// TIA Portal V18 export
TYPE "UDT_RECIPE"
   STRUCT
      TypeName : String[50] := 'Product_1';   // System Defined=
      TypeID : USInt := 1;   // System define= product type for parameters of servo ,press and so on
      FixtureID : Array[1..16] of Byte;
      A1_TableFixtureCode : Array[0..10] of String[128];   // 激光刻印程序号
      A2_TableFixtureCode : Array[0..10] of String[128];   // 贴标10号垂直气缸是否去工作位
      A1RingUnloadingFixtureCode : String[128] := 'SZ23055-OP010-E-Compresspr-ring1 cutting tool';
      E1LoadingNGFixtureCode : String[128] := 'SZ23055-OP010-E-Compressor-Left NG tooling-1';
      ShaftScanFixtureCode : String[128] := 'SZ23055-OP010-E-Compressor-shaft Rotating scanning tooling-1';
      B1PressFixtureCode : String[128] := 'SZ23055-OP010-E-Compressor-ring1 Below Positioning fixture -1';
      CGlueFixtureCode : String[128] := 'SZ23055-OP010-E-Compressor-Point adhesive tooling-1';
      B1PressCylFixtureCode : String[128] := 'SZ23055-OP010-E-Compressor-ring1 Upper pressing fixture-1';
      A2RingUnloadingFixtureCode : String[128] := 'SZ23055-OP010-E-Compresspr-ring2 cutting tool';
      E2UnloadingNGFixtureCode : String[128] := 'SZ23055-OP010-E-Compressor-Right NG tooling-1';
      B2PressFixtureCode : String[128] := 'SZ23055-OP010-E-Compressor-ring2 Below Positioning fixture -1';
      CGlueNGFixtureCode : String[128] := 'SZ23055-OP010-E-Compressor-NG middle shift tooling-1';
      B2PressCylFixtureCode : String[128] := 'SZ23055-OP010-E-Compressor-ring2 Upper pressing fixture-1';
      R1GripperFixtureCode : Array[1..4] of String[128];
      R2GripperFixtureCode : Array[1..4] of String[128];
      R3GripperFixtureCode : Array[1..4] of String[128];
      B1PressProgram : Int := 1;
      B2PressProgram : Int := 1;
      CGlueShaftIV3Program_1 : Word := 16#0001;
      CGlueShaftIV3Program_2 : Word := 16#0002;
      CGlueShaftIV3Program_3 : Word := 16#0003;
      CGlueShaftIV3Program_4 : Word := 16#0004;
      CGlueMagnetIV3Program : Word := 16#0001;
      CGlueProgram : Int := 1;
   END_STRUCT;
   // FixtureID[1] := 16#00;   // 工装编号
   // FixtureID[2..16] := 16#00;
   // A1_TableFixtureCode[0] := '';
   // A1_TableFixtureCode[1] := 'SZ23055-OP010-E-Compressor-ring1 Loading tooling-1';
   // A1_TableFixtureCode[2] := 'SZ23055-OP010-E-Compressor-ring1 Loading tooling-2';
   // A1_TableFixtureCode[3] := 'SZ23055-OP010-E-Compressor-ring1 Loading tooling-3';
   // A1_TableFixtureCode[4] := 'SZ23055-OP010-E-Compressor-ring1 Loading tooling-4';
   // A1_TableFixtureCode[5] := 'SZ23055-OP010-E-Compressor-ring1 Loading tooling-5';
   // A1_TableFixtureCode[6] := 'SZ23055-OP010-E-Compressor-ring1 Loading tooling-6';
   // A1_TableFixtureCode[7] := 'SZ23055-OP010-E-Compressor-ring1 Loading tooling-7';
   // A1_TableFixtureCode[8] := 'SZ23055-OP010-E-Compressor-ring1 Loading tooling-8';
   // A1_TableFixtureCode[9..10] := '';
   // A2_TableFixtureCode[0] := '';
   // A2_TableFixtureCode[1] := 'SZ23055-OP010-E-Compressor-ring2 Loading tooling-1';
   // A2_TableFixtureCode[2] := 'SZ23055-OP010-E-Compressor-ring2 Loading tooling-2';
   // A2_TableFixtureCode[3] := 'SZ23055-OP010-E-Compressor-ring2 Loading tooling-3';
   // A2_TableFixtureCode[4] := 'SZ23055-OP010-E-Compressor-ring2 Loading tooling-4';
   // A2_TableFixtureCode[5] := 'SZ23055-OP010-E-Compressor-ring2 Loading tooling-5';
   // A2_TableFixtureCode[6] := 'SZ23055-OP010-E-Compressor-ring2 Loading tooling-6';
   // A2_TableFixtureCode[7] := 'SZ23055-OP010-E-Compressor-ring2 Loading tooling-7';
   // A2_TableFixtureCode[8] := 'SZ23055-OP010-E-Compressor-ring2 Loading tooling-8';
   // A2_TableFixtureCode[9..10] := '';
   // R1GripperFixtureCode[1] := 'SZ23055-OP010-E-Compressor-robot1 ring1 Left clamping jaw tooling-1';
   // R1GripperFixtureCode[2] := 'SZ23055-OP010-E-Compressor-robot1 ring1 Right clamping jaw tooling-2';
   // R1GripperFixtureCode[3] := 'SZ23055-OP010-E-Compressor-robot1 shaft Left clamping jaw tooling-1';
   // R1GripperFixtureCode[4] := 'SZ23055-OP010-E-Compressor-robot1 shaft Right clamping jaw tooling-2';
   // R2GripperFixtureCode[1] := 'SZ23055-OP010-E-Compressor-robot2 shaft Right clamping jaw tooling-2';
   // R2GripperFixtureCode[2] := 'SZ23055-OP010-E-Compressor-robot2 shaft Left clamping jaw tooling-1';
   // R2GripperFixtureCode[3] := 'SZ23055-OP010-E-Compressor-robot2 magnet Left clamping jaw tooling-1';
   // R2GripperFixtureCode[4] := 'SZ23055-OP010-E-Compressor-robot2 magnet Right clamping jaw tooling-2';
   // R3GripperFixtureCode[1] := 'SZ23055-OP010-E-Compressor-robot3 ring2 Right clamping jaw tooling-2';
   // R3GripperFixtureCode[2] := 'SZ23055-OP010-E-Compressor-robot3 ring2 Left clamping jaw tooling-1';
   // R3GripperFixtureCode[3] := 'SZ23055-OP010-E-Compressor-robot3 shaft Left clamping jaw tooling-1';
   // R3GripperFixtureCode[4] := 'SZ23055-OP010-E-Compressor-robot3 shaft Right clamping jaw tooling-2';
END_TYPE
